FUNCTION_BLOCK DFB_Cylinder
VAR_INPUT
	Sec_P								: BOOL; // One second pulse
	ID									: STRING; // Name that used to logging
	Simulate							: BOOL; // 0: Production mode, 1: Simulation mode
	Permissive							: WORD;
	ShutDown							: WORD;
	AutoInp								: BOOL; // Input command to control cylinder during Auto mode
	Command								: WORD; // Cylinder Command, 1: Retract, 2: Extend, 4: Auto
	IExtend								: BOOL; // Extend feedback signal
	IRetract							: BOOL; // Retract feedback signal
	Travel_Time							: UDINT; // Travel time for cylinder receive extend or retract command
	SetOutput_Pulse						: BOOL;
	FailedHoldLast						: BOOL; // Hold last output command when failed, 0: Not hold, 1: Hold
END_VAR

VAR_OUTPUT
	OExtend								: BOOL; // Extend output signal
	ORetract							: BOOL; // Retract output signal
END_VAR

VAR_IN_OUT
	DUT									: DUT_Cylinder;
END_VAR

VAR
	_Start_up							: BOOL;
	_State_Changed						: BOOL;
	_IExtend							: BOOL;
	_IRetract							: BOOL;
	
	_State								: INT;
	_Last_State							: INT;
	_TLast_State						: INT;
	
	_State_Timer						: UDINT;
	
	_Message							: STRING;
END_VAR

//*********************************************************************************************************************************************************************************************//
// Method Name			: DFB_Cylinder
// Last Modified date	: 25 Feb 2019
// Functionality		: - Handle shut down condition
//						  - Handle reset
//						  - Handle home sensor under simulation mode
//						  - Handle motor condiiton
//						  - Handle motor enable state and EPT
//						  - update target position if not busy
//*********************************************************************************************************************************************************************************************//
// 		Version			Date				Description
//		0.01		21 Feb 2019				Created
//*********************************************************************************************************************************************************************************************//


/////////////////////////////////////////////////////////////////////////////////////////////////////////////////////////////////////////////////////////////////////////////////////////////////
// Start up
/////////////////////////////////////////////////////////////////////////////////////////////////////////////////////////////////////////////////////////////////////////////////////////////////

IF (NOT _Start_up) THEN
	DUT.Enable												:= TRUE;
	_Start_up												:= TRUE;
END_IF

/////////////////////////////////////////////////////////////////////////////////////////////////////////////////////////////////////////////////////////////////////////////////////////////////
// Last Shut Down
/////////////////////////////////////////////////////////////////////////////////////////////////////////////////////////////////////////////////////////////////////////////////////////////////

IF ShutDown <> 0 THEN
	DUT.Last_SD													:= ShutDown;
	DUT.Message													:= F_Concat5(
																	sString1:= CONCAT('Cylinder ID: ', ID), 
																	sString2:= CONCAT(' Shutdown condition triggered: ', WORD_TO_STRING(DUT.Last_SD)), 
																	sString3:= CONCAT('', ''), 
																	sString4:= CONCAT('', ''), 
																	sString5:= CONCAT('', ''));
	Logging.fbDebugLog.M_nLogger(iLogLevel:= iLogVerbosity, sSource:= ' Motor Log ', 
		sMessage												:= DUT.Message);
END_IF


/////////////////////////////////////////////////////////////////////////////////////////////////////////////////////////////////////////////////////////////////////////////////////////////////
// Simulate
/////////////////////////////////////////////////////////////////////////////////////////////////////////////////////////////////////////////////////////////////////////////////////////////////

IF (NOT Simulate) THEN
	_IExtend													:= IExtend;
	_IRetract													:= IRetract;
END_IF


/////////////////////////////////////////////////////////////////////////////////////////////////////////////////////////////////////////////////////////////////////////////////////////////////
// Reset
/////////////////////////////////////////////////////////////////////////////////////////////////////////////////////////////////////////////////////////////////////////////////////////////////

IF DUT.Reset THEN
	DUT.Message													:= '';
	DUT.Failed													:= FALSE;
	DUT.Failed_To_Extend										:= FALSE;
	DUT.Failed_To_Retract										:= FALSE;
	DUT.Reset													:= FALSE;
	_Message													:= F_Concat5(
																	sString1:= CONCAT('Cylinder ID: ', ID), 
																	sString2:= CONCAT(' reset command received: ', ''), 
																	sString3:= CONCAT('', ''), 
																	sString4:= CONCAT('', ''), 
																	sString5:= CONCAT('', ''));
	Logging.fbDebugLog.M_nLogger(iLogLevel:= iLogVerbosity, sSource:= ' Motor Log ', 
		sMessage												:= _Message);
END_IF


/////////////////////////////////////////////////////////////////////////////////////////////////////////////////////////////////////////////////////////////////////////////////////////////////
// Status
/////////////////////////////////////////////////////////////////////////////////////////////////////////////////////////////////////////////////////////////////////////////////////////////////

// Enable state
IF DUT.Enable THEN
	DUT.EnbState												:= Enum_ModuleEnableState.eEnabled;
ELSE
	DUT.EnbState												:= Enum_ModuleEnableState.eDisabled;
END_IF

// EPT 
IF DUT.Failed OR DUT.CMD <> 4 OR (NOT DUT.Enable) OR DUT.Callibration_Mode THEN
	DUT.EPT														:= Enum_EPT.eBlocked;
ELSIF _State = 10 OR _State = 20 THEN
	DUT.EPT														:= Enum_EPT.eBusy;
ELSE
	DUT.EPT														:= Enum_EPT.eIdle;
END_IF

// Status
IF DUT.Failed THEN
	DUT.Status													:= 99;
ELSIF _IRetract THEN
	DUT.Status													:= 1;
ELSIF _IExtend THEN
	DUT.Status													:= 2;
END_IF


/////////////////////////////////////////////////////////////////////////////////////////////////////////////////////////////////////////////////////////////////////////////////////////////////
// Cyclic call
/////////////////////////////////////////////////////////////////////////////////////////////////////////////////////////////////////////////////////////////////////////////////////////////////

SEQ();


/////////////////////////////////////////////////////////////////////////////////////////////////////////////////////////////////////////////////////////////////////////////////////////////////
// Mapping
/////////////////////////////////////////////////////////////////////////////////////////////////////////////////////////////////////////////////////////////////////////////////////////////////

DUT.Failed														:= DUT.Failed_To_Extend OR DUT.Failed_To_Retract OR DUT.Failed;
DUT.CylinderID													:= ID;
DUT.Simulate													:= Simulate;
DUT.Enable														:= DUT.Enable;

DUT.Extended													:= IExtend;
DUT.Retracted													:= IRetract;

ACTION SEQ:
//////////////////////////////////////////////////////////////////////////////////////////////////////////////////////////////////////////////////////////////////
// State timer
//////////////////////////////////////////////////////////////////////////////////////////////////////////////////////////////////////////////////////////////////

_State_Changed													:= _TLast_State <> _State;
_TLast_State													:= _State;

IF _State_Changed THEN
	_State_Timer												:= 0;
	_Message													:= F_Concat5(
																	sString1:= CONCAT('Cylinder ID: ', ID), 
																	sString2:= CONCAT(', Current state: ', INT_TO_STRING(_State)), 
																	sString3:= CONCAT('', ''), 
																	sString4:= CONCAT('', ''), 
																	sString5:= CONCAT('', ''));
	Logging.fbDebugLog.M_nLogger(iLogLevel:= iLogVerbosity, sSource:= ' DFB_Cylinder.SEQ ', 
		sMessage												:= _Message);
ELSE
	IF Sec_P THEN
		_State_Timer											:= _State_Timer + 1;
	END_IF
END_IF


//////////////////////////////////////////////////////////////////////////////////////////////////////////////////////////////////////////////////////////////////
// State machine
//////////////////////////////////////////////////////////////////////////////////////////////////////////////////////////////////////////////////////////////////

CASE _State OF
	0: (*Idle*)
		
		(*Action*)
		OExtend													:= FALSE;
		ORetract												:= FALSE;
		
		(*Transition*)
		IF Permissive = 16#FFFF THEN
			_State												:= 1; // Ready
		ELSIF DUT.CMD = 1 OR DUT.CMD = 2 OR (DUT.CMD = 4 AND AutoInp) THEN
			DUT.Message											:= F_Concat5(
																	sString1:= CONCAT('Cylinder ID: ', ID), 
																	sString2:= CONCAT(' permissive not fulfill - ', WORD_TO_STRING(Permissive)), 
																	sString3:= CONCAT('', ''), 
																	sString4:= CONCAT('', ''), 
																	sString5:= CONCAT('', ''));
			DUT.Failed											:= TRUE;
			_State												:= 99; // Error
		END_IF
		
	1: (*Ready*)
		_Last_State												:= 1;
	
		(*Action*)
		
		(*Transition*)
		IF (DUT.CMD = 2 OR (DUT.CMD = 4 AND AutoInp)) AND ((NOT IExtend) OR (NOT OExtend AND (NOT SetOutput_Pulse))) THEN
			_State												:= 10; // Extending
		ELSIF (DUT.CMD = 1 OR (DUT.CMD = 4 AND (NOT AutoInp))) AND ((NOT IRetract) OR (NOT ORetract AND (NOT SetOutput_Pulse))) THEN
			_State												:= 20; // Retracting
		END_IF
	
	10: (*Extending*)
		_Last_State												:= 10;
	
		(*Action*)
		OExtend													:= TRUE;
		ORetract												:= FALSE;
		
		IF Simulate THEN
			_IExtend											:= TRUE;
			_IRetract											:= FALSE;
		END_IF
		
		(*Transition*)
		IF ShutDown = 0 THEN
			IF DUT.CMD = 1 OR (DUT.CMD = 4 AND (NOT AutoInp)) THEN
				_State											:= 20; // Retracting
			ELSIF _State_Timer > 1 THEN
				IF _IExtend THEN
					_State										:= 11; // Extended
				ELSIF _State_Timer > Travel_Time THEN
					DUT.Failed_To_Extend						:= TRUE;
					DUT.Message									:= F_Concat5(
																	sString1:= CONCAT('Cylinder ID: ', ID), 
																	sString2:= CONCAT(' failed to receive extend feedback signal', ''), 
																	sString3:= CONCAT('', ''), 
																	sString4:= CONCAT('', ''), 
																	sString5:= CONCAT('', ''));
					Logging.fbDebugLog.M_nLogger(iLogLevel:= iLogVerbosity, sSource:= ' Motor Log ', 
						sMessage								:= DUT.Message);
					_State										:= 99; // Error
				END_IF
			END_IF
		ELSE
			DUT.Failed											:= TRUE;
			_State												:= 99; // Error
		END_IF
		
	
	11: (*Extended*)
		_Last_State												:= 11;
	
		(*Action*)
		IF SetOutput_Pulse THEN
			OExtend												:= FALSE;
			ORetract											:= FALSE;
		ELSE
			OExtend												:= TRUE;
			ORetract											:= FALSE;
		END_IF
		
		(*Transition*)
		IF ShutDown = 0 THEN
			IF DUT.CMD = 1 OR (DUT.CMD = 4 AND (NOT AutoInp)) THEN
				_State											:= 20; // Retracting
			ELSIF (NOT _IExtend) THEN
				DUT.Failed_To_Extend							:= TRUE;
				_State											:= 99;
			END_IF
		ELSE
			DUT.Failed											:= TRUE;
			_State												:= 99; // Error
		END_IF
	
	20: (*Retracting*)
		_Last_State												:= 20;
	
		(*Action*)
		OExtend													:= FALSE;
		ORetract												:= TRUE;
		
		IF Simulate THEN
			_IExtend											:= FALSE;
			_IRetract											:= TRUE;
		END_IF
		
		(*Transition*)
		IF ShutDown = 0 THEN
			IF DUT.CMD = 2 OR (DUT.CMD = 4 AND AutoInp) THEN
				_State											:= 10; // Retracting
			ELSIF _State_Timer > 1 THEN
				IF _IRetract THEN
					_State										:= 21; // Retracted
				ELSIF _State_Timer > Travel_Time THEN
					DUT.Failed_To_Retract						:= TRUE;
					DUT.Message									:= F_Concat5(
																	sString1:= CONCAT('Cylinder ID: ', ID), 
																	sString2:= CONCAT(' failed to receive retract feedback signal', ''), 
																	sString3:= CONCAT('', ''), 
																	sString4:= CONCAT('', ''), 
																	sString5:= CONCAT('', ''));
					Logging.fbDebugLog.M_nLogger(iLogLevel:= iLogVerbosity, sSource:= ' Motor Log ', 
						sMessage								:= DUT.Message);
					_State										:= 99; // Error
				END_IF
			END_IF
		ELSE
			DUT.Failed											:= TRUE;
			_State												:= 99; // Error
		END_IF
	
	21: (*Retracted*)
		_Last_State												:= 21;
	
		(*Action*)
		IF SetOutput_Pulse THEN
			OExtend												:= FALSE;
			ORetract											:= FALSE;
		ELSE
			OExtend												:= FALSE;
			ORetract											:= TRUE;
		END_IF
		
		(*Transition*)
		IF ShutDown = 0 THEN
			IF DUT.CMD = 2 OR (DUT.CMD = 4 AND AutoInp) THEN
				_State											:= 10; // Retracting
			ELSIF (NOT _IRetract) THEN
				DUT.Failed_To_Retract							:= TRUE;
				_State											:= 99; 
			END_IF
		ELSE
			DUT.Failed											:= TRUE;
			_State												:= 99; // Error
		END_IF
		
	99: (*Error*)
	
		(*Action*)
		IF FailedHoldLast THEN
			OExtend												:= OExtend;
			ORetract											:= ORetract;
		ELSE	
			OExtend												:= FALSE;
			ORetract											:= FALSE;
		END_IF
	
		(*Transition*)
		IF (NOT DUT.Failed) THEN
			_State												:= 0; // Idle
		END_IF
END_CASE
END_ACTION

END_FUNCTION_BLOCK

(* stored: Version 1.1.0.1, ProductVersion 3.1.4022.18
   POU DFB_Cylinder: Id {d48d630f-3ffe-4d0a-a1ab-d31f442126fc}, SpecialFunc None
   Action SEQ: Id {26e7a909-86c7-4852-9018-cb8b44a72c81} *)
